PROGRAM MAIN
VAR
END_VAR

END_PROGRAM

(* stored: Version 1.1.0.1, ProductVersion 3.1.0.12
   POU MAIN: Id {f59074d3-ce33-48d0-9823-d5ddf0b28bf1} *)
